PROGRAM Control
VAR


	ToggleSpiral: TOGGLE;
	HopperLevel_High: TON;
	HopperLevelHigh: BOOL;
	HopperLevelLow: BOOL;
	HopperLevelISLow: BOOL;
	HopperLevelISHigh: BOOL;
	Hopper_Level: Hopper_Level;
	Hopper_LevelLow: TON;
	Twin_Auger_Level: Hopper_Level;
	FRA3_HopperLevel_INT: INT;
	sSpice_Tank_Valve: BOOL;
	PreBrine_Delay: TON;
	PreBrineValveTON: TON;
	PreBrineValveTOF: TOF;
	Feed: ton;
	Auger: ton;
	FeedAugerResume: ton;
	Resume: BOOL;
	Auger_Resume: BOOL;
	HopperResume: tof;
	FillerCPM: FillerCPM_Current;
	sFillerCPM_Current: REAL;
	HopperLevelLow_Timer: TIME;
	SpareTON_1: TON;
END_VAR
VAR PERSISTENT
	SpareTONTest: BOOL;
	SpareTimerTest: BOOL;
	HopperLevelLowHMI: INT;
	HopperLevelLowCalc: INT;
	HopperLevelHighHMI: INT;
	HopperLevelHighCalc: INT;
	HopperLevelHigh_Timer: TIME;
	FeedAugerResumeHMI: INT;
	FeedAugerResumeCalc: INT;
	FeedAugerDelayHMITimer: TIME;
	sCloserJam_1_RealValue: REAL;
	sCloserJam_1RV: REAL;
	sCloserJam_1PT: TIME;
	sCloserJam_2_RealValue: REAL;
	sCloserJam_2RV: REAL;
	sCloserJam_2PT: TIME;
	sElevatorJam_RealValue: REAL;
	sElevatorJamRV: REAL;
	sElevatorJamPT: TIME;
	sFullCanBeltDelay_RealValue: REAL;
	sFullCanBeltDelayRV: REAL;
	sFullCanBeltDelayPT: TIME;
	sNoEmptyCansDelay_RealValue: REAL;
	sNoEmptyCansDelayRV: REAL;
	sNoEmptyCansDelayPT: TIME;
	sPrebrineFlapON_RealValue: REAL;
	sPrebrineFlapOFFRV: REAL;
	sPrebrineFlapONRV: REAL;
	sPrebrineFlapONPT: TIME;
	sPrebrineFlapOFF_RealValue: REAL;
	sPrebrineFlapOFFPT: TIME;
	sPrebrineValveON_RealValue: REAL;
	sPrebrineValveONRV: REAL;
	sPrebrineValveONPT: TIME;
	sPrebrineValveOFF_RealValue: REAL;
	sPrebrineValveOffRV: REAL;
	sPrebrineValveOffPT: TIME;
	sRefillJuicer_RealValue: REAL;
	sRefillJuicerRV: REAL;
	sRefillJuicerPT: TIME;
	sLowSpiceDisable_RealValue: REAL;
	sLowSpiceDisableRV: REAL;
	sLowSpiceDisablePT: TIME;
END_VAR
VAR // added by the converter: edge detectors and wires of the graphical bodies
    _w1, _w2, _w3 : BOOL;
END_VAR

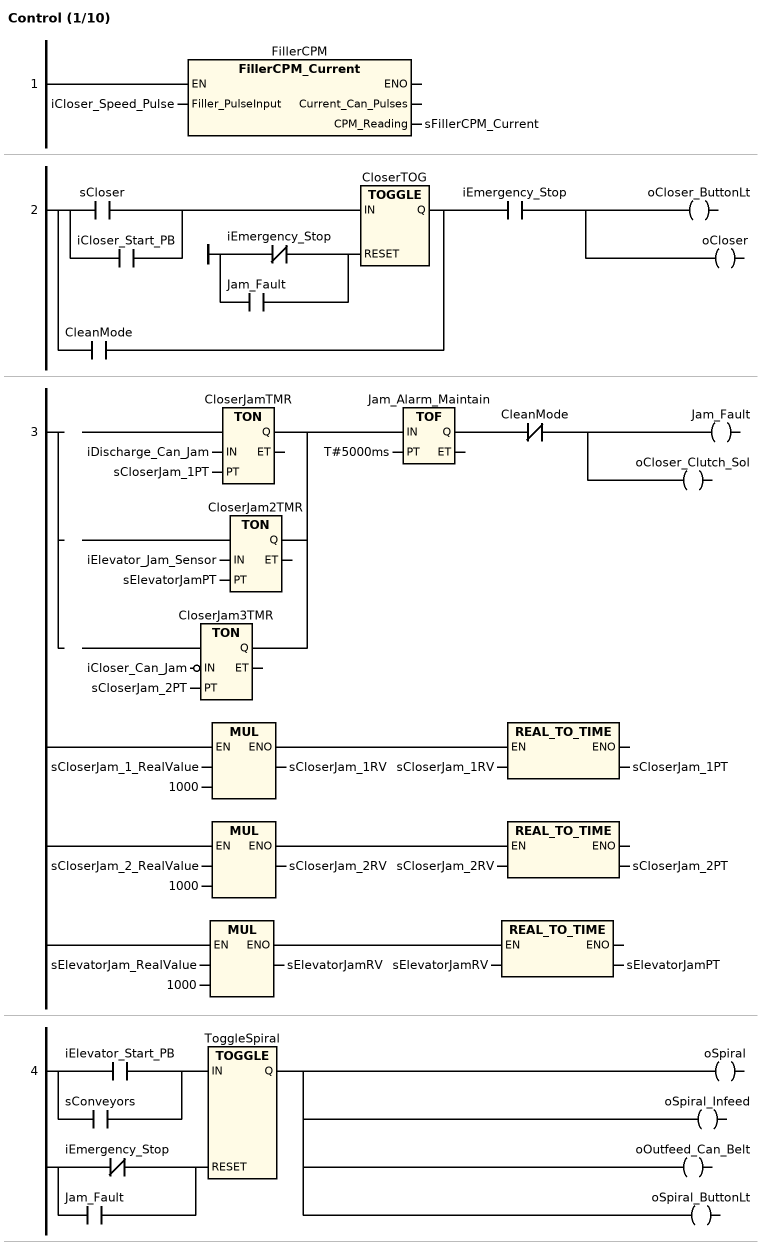
// NETWORK 1
FillerCPM(Filler_PulseInput := iCloser_Speed_Pulse, CPM_Reading => sFillerCPM_Current); // FillerCPM_Current

// NETWORK 2
CloserTOG(IN := sCloser OR iCloser_Start_PB, RESET := NOT iEmergency_Stop OR Jam_Fault); // TOGGLE
_w1 := (CloserTOG.Q OR CleanMode) AND iEmergency_Stop;
oCloser_ButtonLt := _w1;
oCloser := _w1;

// NETWORK 3
CloserJamTMR(IN := iDischarge_Can_Jam, PT := sCloserJam_1PT); // TON
CloserJam2TMR(IN := iElevator_Jam_Sensor, PT := sElevatorJamPT); // TON
CloserJam3TMR(IN := NOT iCloser_Can_Jam, PT := sCloserJam_2PT); // TON
Jam_Alarm_Maintain(IN := CloserJamTMR.Q OR CloserJam2TMR.Q OR CloserJam3TMR.Q, PT := T#5000ms); // TOF
_w2 := Jam_Alarm_Maintain.Q AND NOT CleanMode;
Jam_Fault := _w2;
oCloser_Clutch_Sol := _w2;
sCloserJam_1RV := sCloserJam_1_RealValue * 1000;
sCloserJam_1PT := REAL_TO_TIME(sCloserJam_1RV);
sCloserJam_2RV := sCloserJam_2_RealValue * 1000;
sCloserJam_2PT := REAL_TO_TIME(sCloserJam_2RV);
sElevatorJamRV := sElevatorJam_RealValue * 1000;
sElevatorJamPT := REAL_TO_TIME(sElevatorJamRV);

// NETWORK 4
ToggleSpiral(IN := iElevator_Start_PB OR sConveyors, RESET := NOT iEmergency_Stop OR Jam_Fault); // TOGGLE
oSpiral := ToggleSpiral.Q;
oSpiral_Infeed := ToggleSpiral.Q;
oOutfeed_Can_Belt := ToggleSpiral.Q;
oSpiral_ButtonLt := ToggleSpiral.Q;

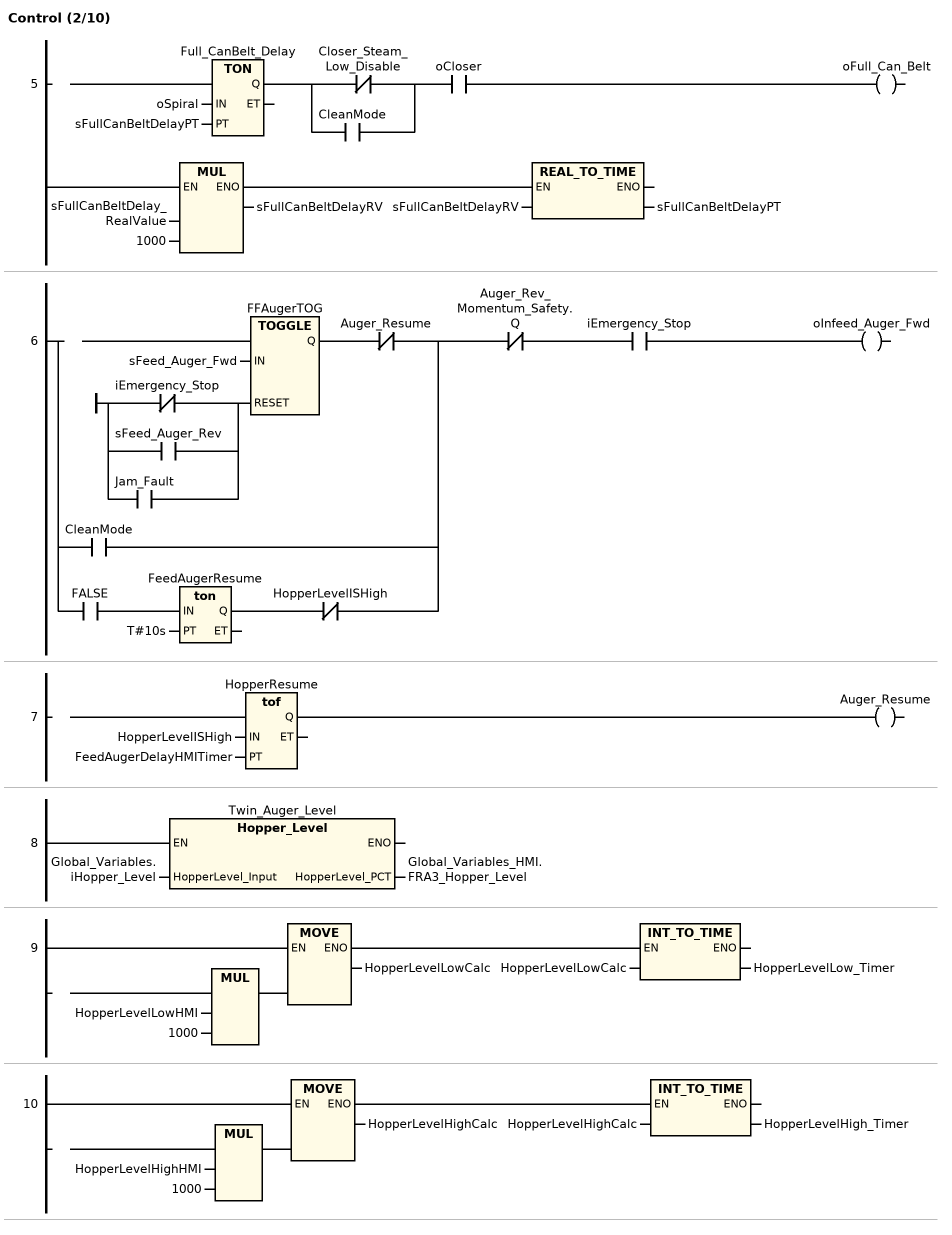
// NETWORK 5
Full_CanBelt_Delay(IN := oSpiral, PT := sFullCanBeltDelayPT); // TON
oFull_Can_Belt := Full_CanBelt_Delay.Q AND (NOT Closer_Steam_Low_Disable OR CleanMode) AND oCloser;
sFullCanBeltDelayRV := sFullCanBeltDelay_RealValue * 1000;
sFullCanBeltDelayPT := REAL_TO_TIME(sFullCanBeltDelayRV);

// NETWORK 6
FFAugerTOG(IN := sFeed_Auger_Fwd, RESET := NOT iEmergency_Stop OR sFeed_Auger_Rev OR Jam_Fault); // TOGGLE
FeedAugerResume(IN := FALSE, PT := T#10s); // ton
oInfeed_Auger_Fwd := (FFAugerTOG.Q AND NOT Auger_Resume OR CleanMode OR FeedAugerResume.Q AND NOT HopperLevelISHigh) AND NOT Auger_Rev_Momentum_Safety.Q AND iEmergency_Stop;

// NETWORK 7
HopperResume(IN := HopperLevelISHigh, PT := FeedAugerDelayHMITimer); // tof
Auger_Resume := HopperResume.Q;

// NETWORK 8
Twin_Auger_Level(HopperLevel_Input := Global_Variables.iHopper_Level, HopperLevel_PCT => Global_Variables_HMI.FRA3_Hopper_Level); // Hopper_Level

// NETWORK 9
HopperLevelLowCalc := HopperLevelLowHMI * 1000;
HopperLevelLow_Timer := INT_TO_TIME(HopperLevelLowCalc);

// NETWORK 10
HopperLevelHighCalc := HopperLevelHighHMI * 1000;
HopperLevelHigh_Timer := INT_TO_TIME(HopperLevelHighCalc);

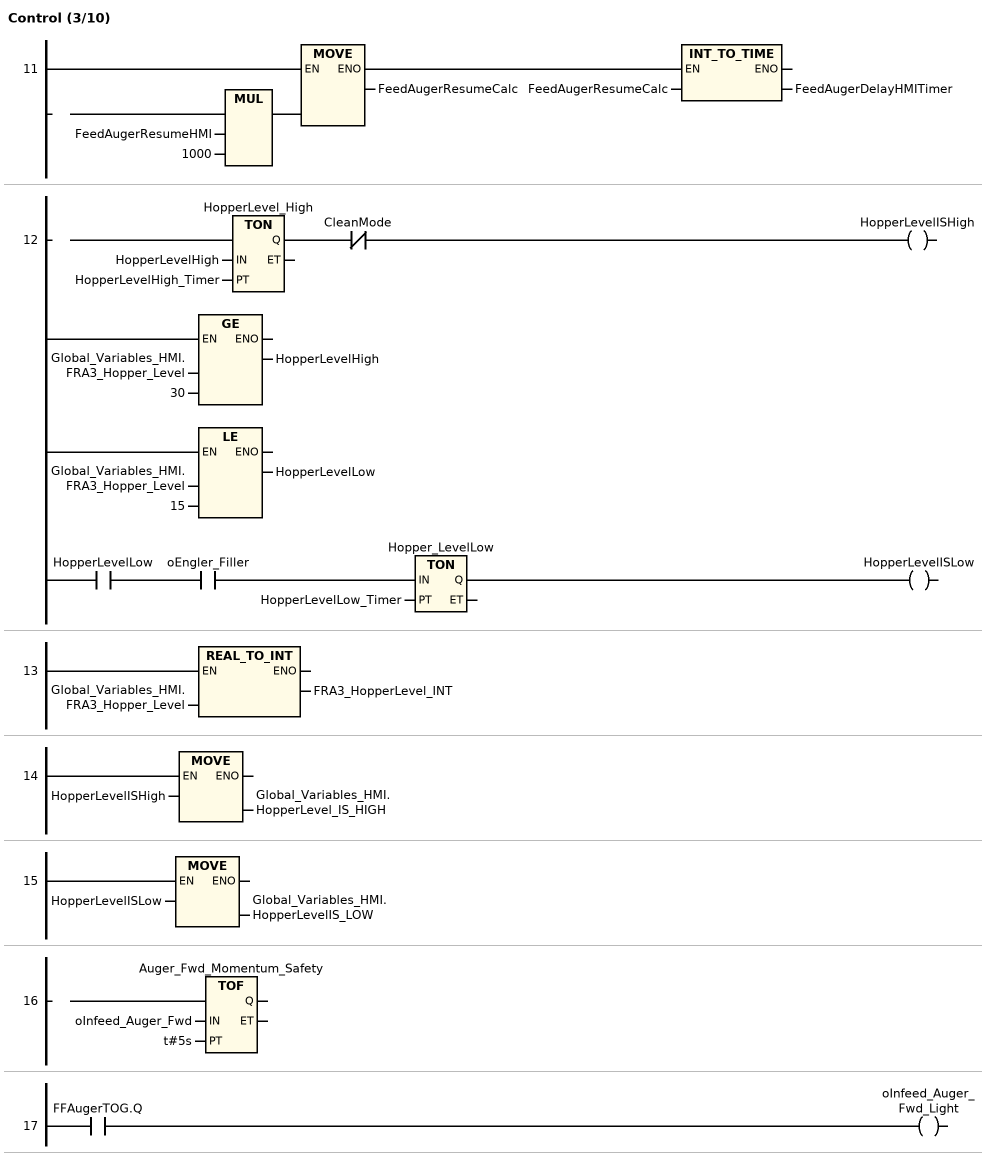
// NETWORK 11
FeedAugerResumeCalc := FeedAugerResumeHMI * 1000;
FeedAugerDelayHMITimer := INT_TO_TIME(FeedAugerResumeCalc);

// NETWORK 12
HopperLevel_High(IN := HopperLevelHigh, PT := HopperLevelHigh_Timer); // TON
HopperLevelISHigh := HopperLevel_High.Q AND NOT CleanMode;
HopperLevelHigh := Global_Variables_HMI.FRA3_Hopper_Level >= 30;
HopperLevelLow := Global_Variables_HMI.FRA3_Hopper_Level <= 15;
Hopper_LevelLow(IN := HopperLevelLow AND oEngler_Filler, PT := HopperLevelLow_Timer); // TON
HopperLevelISLow := Hopper_LevelLow.Q;

// NETWORK 13
FRA3_HopperLevel_INT := REAL_TO_INT(Global_Variables_HMI.FRA3_Hopper_Level);

// NETWORK 14
Global_Variables_HMI.HopperLevel_IS_HIGH := HopperLevelISHigh;

// NETWORK 15
Global_Variables_HMI.HopperLevelIS_LOW := HopperLevelISLow;

// NETWORK 16
Auger_Fwd_Momentum_Safety(IN := oInfeed_Auger_Fwd, PT := t#5s); // TOF

// NETWORK 17
oInfeed_Auger_Fwd_Light := FFAugerTOG.Q;

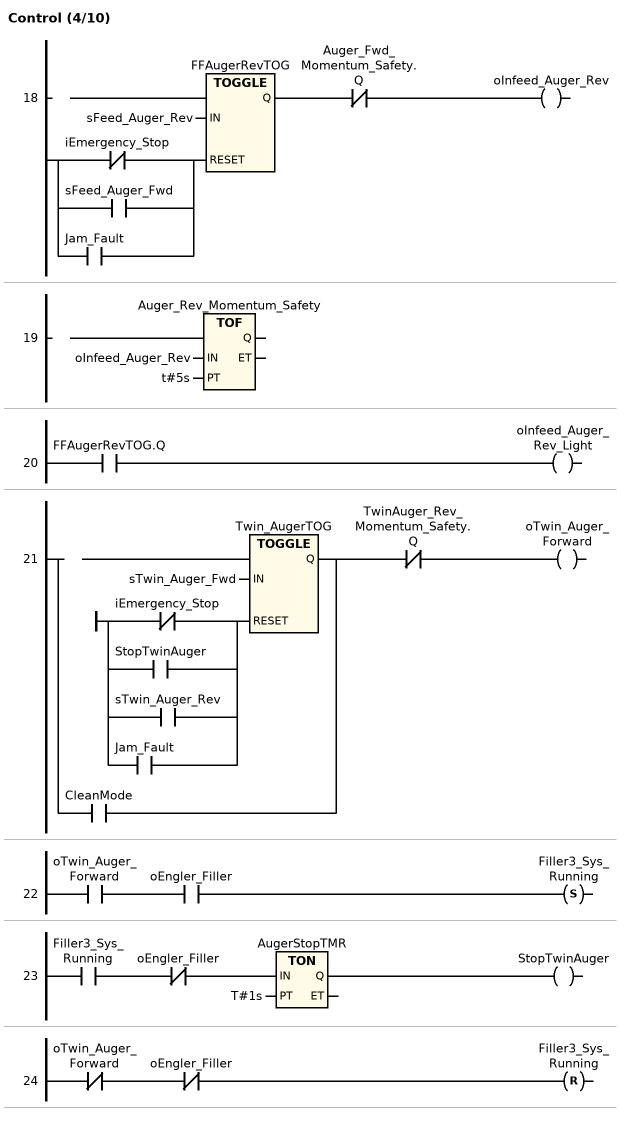
// NETWORK 18
FFAugerRevTOG(IN := sFeed_Auger_Rev, RESET := NOT iEmergency_Stop OR sFeed_Auger_Fwd OR Jam_Fault); // TOGGLE
oInfeed_Auger_Rev := FFAugerRevTOG.Q AND NOT Auger_Fwd_Momentum_Safety.Q;

// NETWORK 19
Auger_Rev_Momentum_Safety(IN := oInfeed_Auger_Rev, PT := t#5s); // TOF

// NETWORK 20
oInfeed_Auger_Rev_Light := FFAugerRevTOG.Q;

// NETWORK 21
Twin_AugerTOG(IN := sTwin_Auger_Fwd, RESET := NOT iEmergency_Stop OR StopTwinAuger OR sTwin_Auger_Rev OR Jam_Fault); // TOGGLE
oTwin_Auger_Forward := (Twin_AugerTOG.Q OR CleanMode) AND NOT TwinAuger_Rev_Momentum_Safety.Q;

// NETWORK 22
Filler3_Sys_Running S= oTwin_Auger_Forward AND oEngler_Filler;

// NETWORK 23
AugerStopTMR(IN := Filler3_Sys_Running AND NOT oEngler_Filler, PT := T#1s); // TON
StopTwinAuger := AugerStopTMR.Q;

// NETWORK 24
Filler3_Sys_Running R= NOT oTwin_Auger_Forward AND NOT oEngler_Filler;

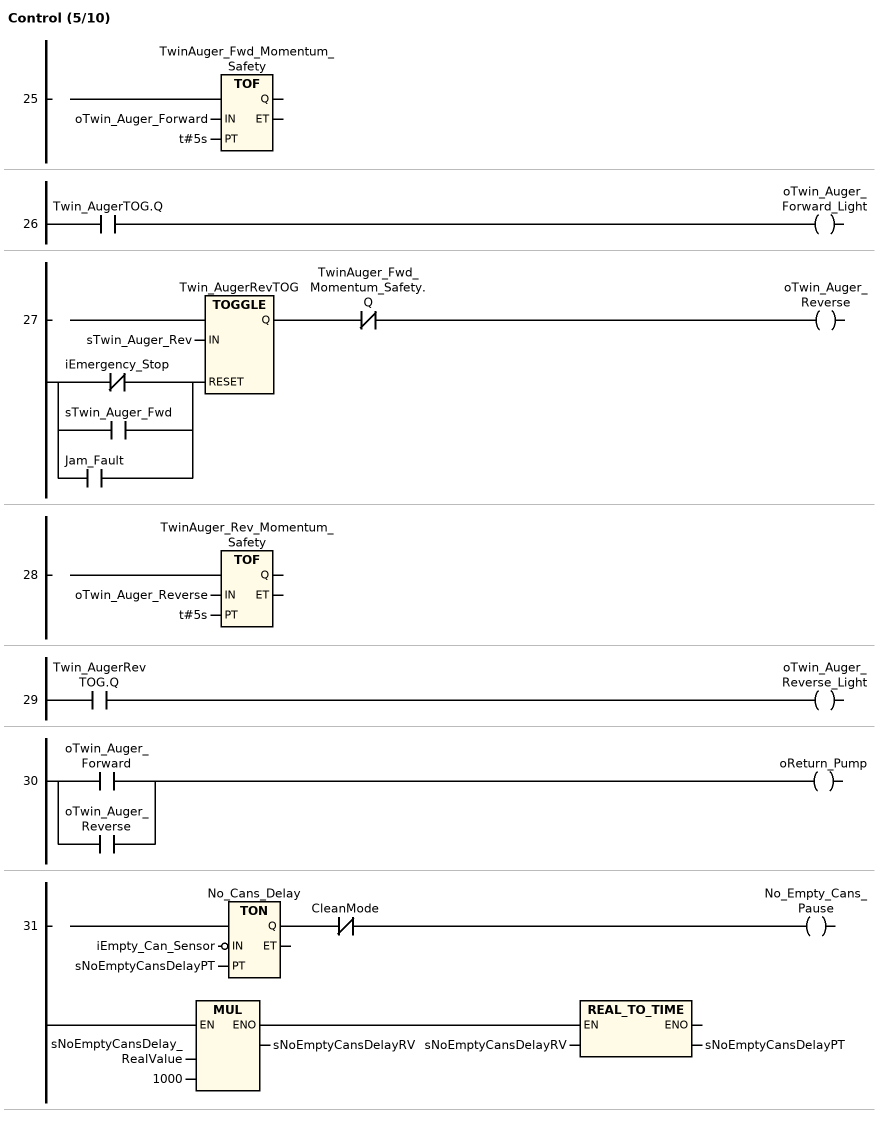
// NETWORK 25
TwinAuger_Fwd_Momentum_Safety(IN := oTwin_Auger_Forward, PT := t#5s); // TOF

// NETWORK 26
oTwin_Auger_Forward_Light := Twin_AugerTOG.Q;

// NETWORK 27
Twin_AugerRevTOG(IN := sTwin_Auger_Rev, RESET := NOT iEmergency_Stop OR sTwin_Auger_Fwd OR Jam_Fault); // TOGGLE
oTwin_Auger_Reverse := Twin_AugerRevTOG.Q AND NOT TwinAuger_Fwd_Momentum_Safety.Q;

// NETWORK 28
TwinAuger_Rev_Momentum_Safety(IN := oTwin_Auger_Reverse, PT := t#5s); // TOF

// NETWORK 29
oTwin_Auger_Reverse_Light := Twin_AugerRevTOG.Q;

// NETWORK 30
oReturn_Pump := oTwin_Auger_Forward OR oTwin_Auger_Reverse;

// NETWORK 31
No_Cans_Delay(IN := NOT iEmpty_Can_Sensor, PT := sNoEmptyCansDelayPT); // TON
No_Empty_Cans_Pause := No_Cans_Delay.Q AND NOT CleanMode;
sNoEmptyCansDelayRV := sNoEmptyCansDelay_RealValue * 1000;
sNoEmptyCansDelayPT := REAL_TO_TIME(sNoEmptyCansDelayRV);

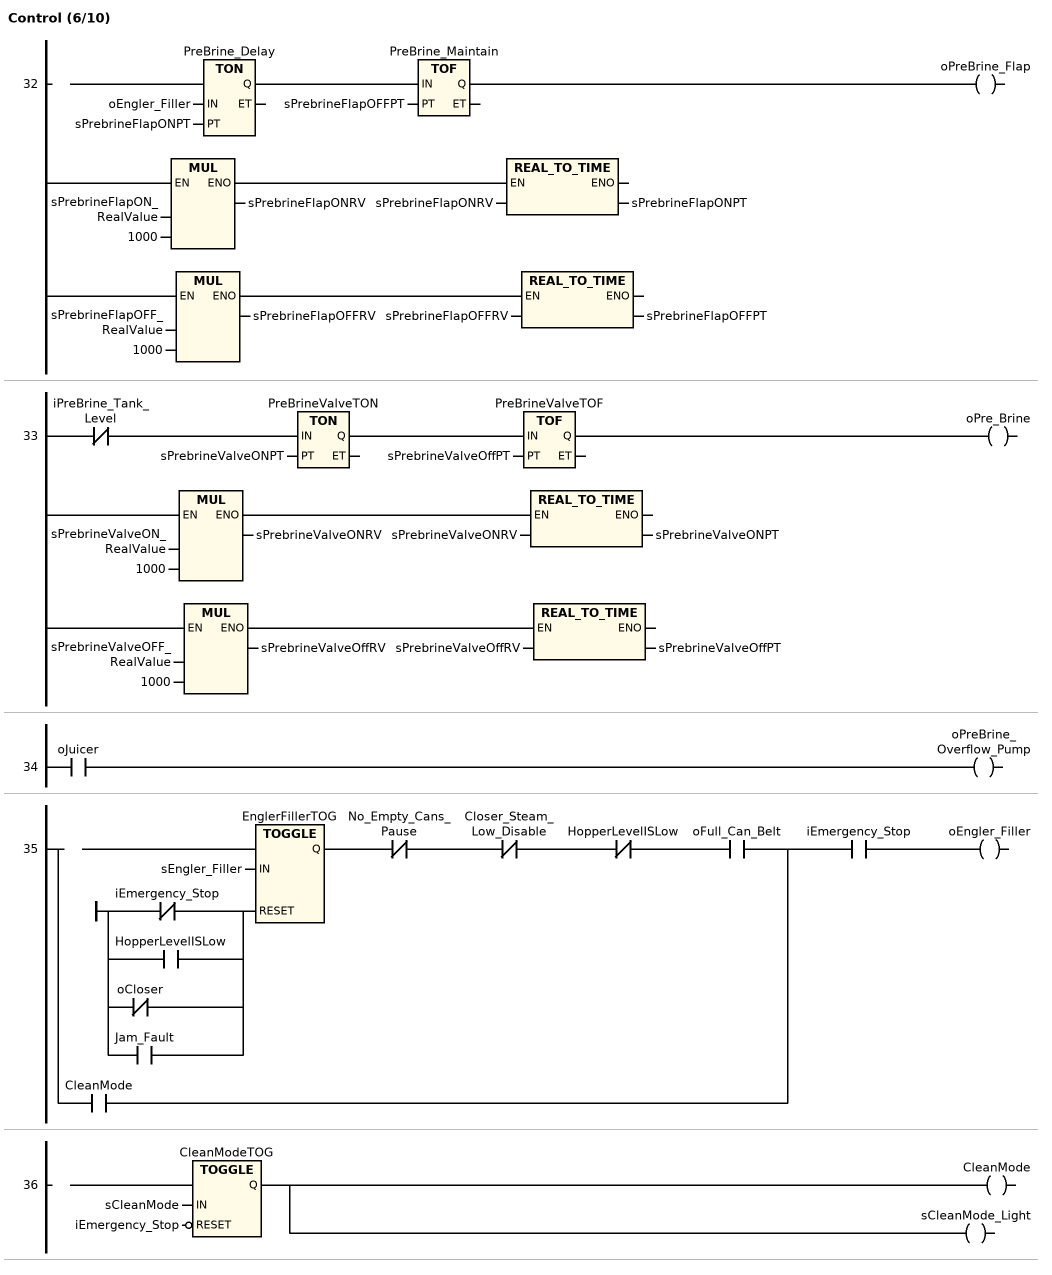
// NETWORK 32
PreBrine_Delay(IN := oEngler_Filler, PT := sPrebrineFlapONPT); // TON
PreBrine_Maintain(IN := PreBrine_Delay.Q, PT := sPrebrineFlapOFFPT); // TOF
oPreBrine_Flap := PreBrine_Maintain.Q;
sPrebrineFlapONRV := sPrebrineFlapON_RealValue * 1000;
sPrebrineFlapONPT := REAL_TO_TIME(sPrebrineFlapONRV);
sPrebrineFlapOFFRV := sPrebrineFlapOFF_RealValue * 1000;
sPrebrineFlapOFFPT := REAL_TO_TIME(sPrebrineFlapOFFRV);

// NETWORK 33
PreBrineValveTON(IN := NOT iPreBrine_Tank_Level, PT := sPrebrineValveONPT); // TON
PreBrineValveTOF(IN := PreBrineValveTON.Q, PT := sPrebrineValveOffPT); // TOF
oPre_Brine := PreBrineValveTOF.Q;
sPrebrineValveONRV := sPrebrineValveON_RealValue * 1000;
sPrebrineValveONPT := REAL_TO_TIME(sPrebrineValveONRV);
sPrebrineValveOffRV := sPrebrineValveOFF_RealValue * 1000;
sPrebrineValveOffPT := REAL_TO_TIME(sPrebrineValveOffRV);

// NETWORK 34
oPreBrine_Overflow_Pump := oJuicer;

// NETWORK 35
EnglerFillerTOG(IN := sEngler_Filler, RESET := NOT iEmergency_Stop OR HopperLevelISLow OR NOT oCloser OR Jam_Fault); // TOGGLE
oEngler_Filler := (EnglerFillerTOG.Q AND NOT No_Empty_Cans_Pause AND NOT Closer_Steam_Low_Disable AND NOT HopperLevelISLow AND oFull_Can_Belt OR CleanMode) AND iEmergency_Stop;

// NETWORK 36
CleanModeTOG(IN := sCleanMode, RESET := NOT iEmergency_Stop); // TOGGLE
CleanMode := CleanModeTOG.Q;
sCleanMode_Light := CleanModeTOG.Q;

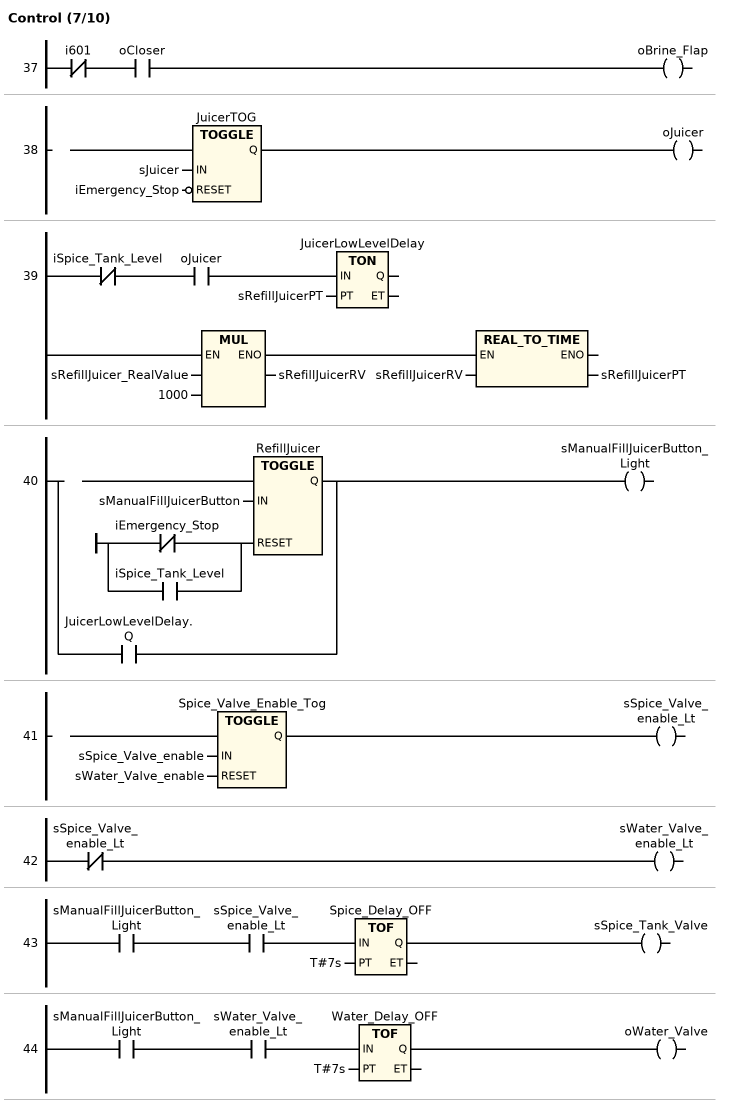
// NETWORK 37
oBrine_Flap := NOT i601 AND oCloser;

// NETWORK 38
JuicerTOG(IN := sJuicer, RESET := NOT iEmergency_Stop); // TOGGLE
oJuicer := JuicerTOG.Q;

// NETWORK 39
JuicerLowLevelDelay(IN := NOT iSpice_Tank_Level AND oJuicer, PT := sRefillJuicerPT); // TON
sRefillJuicerRV := sRefillJuicer_RealValue * 1000;
sRefillJuicerPT := REAL_TO_TIME(sRefillJuicerRV);

// NETWORK 40
RefillJuicer(IN := sManualFillJuicerButton, RESET := NOT iEmergency_Stop OR iSpice_Tank_Level); // TOGGLE
sManualFillJuicerButton_Light := RefillJuicer.Q OR JuicerLowLevelDelay.Q;

// NETWORK 41
Spice_Valve_Enable_Tog(IN := sSpice_Valve_enable, RESET := sWater_Valve_enable); // TOGGLE
sSpice_Valve_enable_Lt := Spice_Valve_Enable_Tog.Q;

// NETWORK 42
sWater_Valve_enable_Lt := NOT sSpice_Valve_enable_Lt;

// NETWORK 43
Spice_Delay_OFF(IN := sManualFillJuicerButton_Light AND sSpice_Valve_enable_Lt, PT := T#7s); // TOF
sSpice_Tank_Valve := Spice_Delay_OFF.Q;

// NETWORK 44
Water_Delay_OFF(IN := sManualFillJuicerButton_Light AND sWater_Valve_enable_Lt, PT := T#7s); // TOF
oWater_Valve := Water_Delay_OFF.Q;

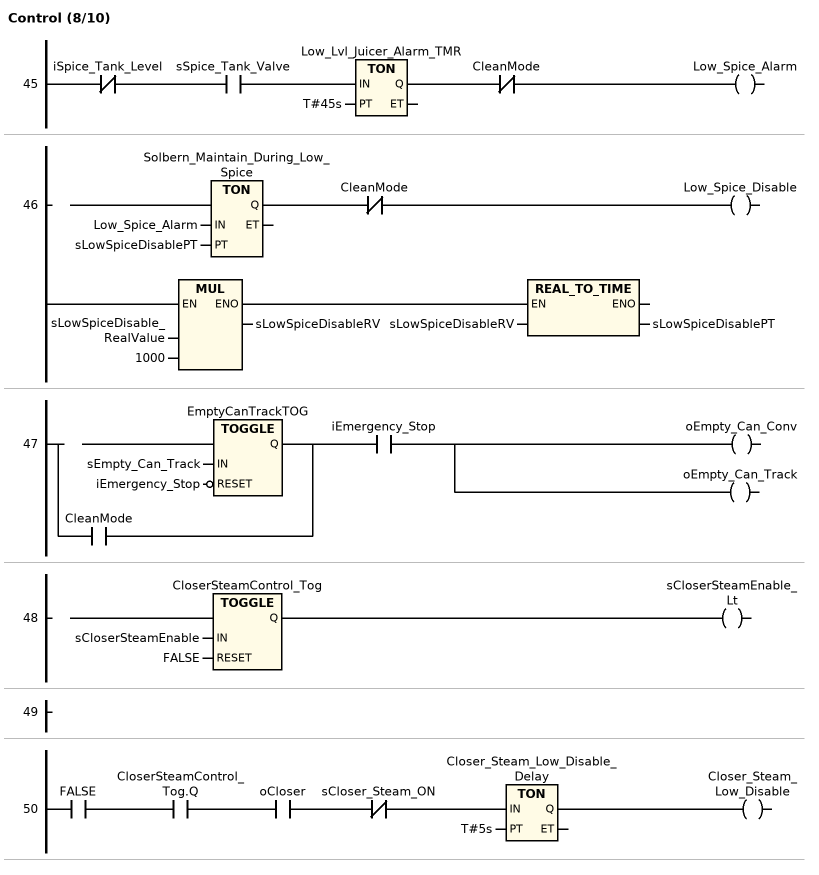
// NETWORK 45
Low_Lvl_Juicer_Alarm_TMR(IN := NOT iSpice_Tank_Level AND sSpice_Tank_Valve, PT := T#45s); // TON
Low_Spice_Alarm := Low_Lvl_Juicer_Alarm_TMR.Q AND NOT CleanMode;

// NETWORK 46
Solbern_Maintain_During_Low_Spice(IN := Low_Spice_Alarm, PT := sLowSpiceDisablePT); // TON
Low_Spice_Disable := Solbern_Maintain_During_Low_Spice.Q AND NOT CleanMode;
sLowSpiceDisableRV := sLowSpiceDisable_RealValue * 1000;
sLowSpiceDisablePT := REAL_TO_TIME(sLowSpiceDisableRV);

// NETWORK 47
EmptyCanTrackTOG(IN := sEmpty_Can_Track, RESET := NOT iEmergency_Stop); // TOGGLE
_w3 := (EmptyCanTrackTOG.Q OR CleanMode) AND iEmergency_Stop;
oEmpty_Can_Conv := _w3;
oEmpty_Can_Track := _w3;

// NETWORK 48
CloserSteamControl_Tog(IN := sCloserSteamEnable, RESET := FALSE); // TOGGLE
sCloserSteamEnable_Lt := CloserSteamControl_Tog.Q;

// NETWORK 49

// NETWORK 50
Closer_Steam_Low_Disable_Delay(IN := FALSE AND CloserSteamControl_Tog.Q AND oCloser AND NOT sCloser_Steam_ON, PT := T#5s); // TON
Closer_Steam_Low_Disable := Closer_Steam_Low_Disable_Delay.Q;

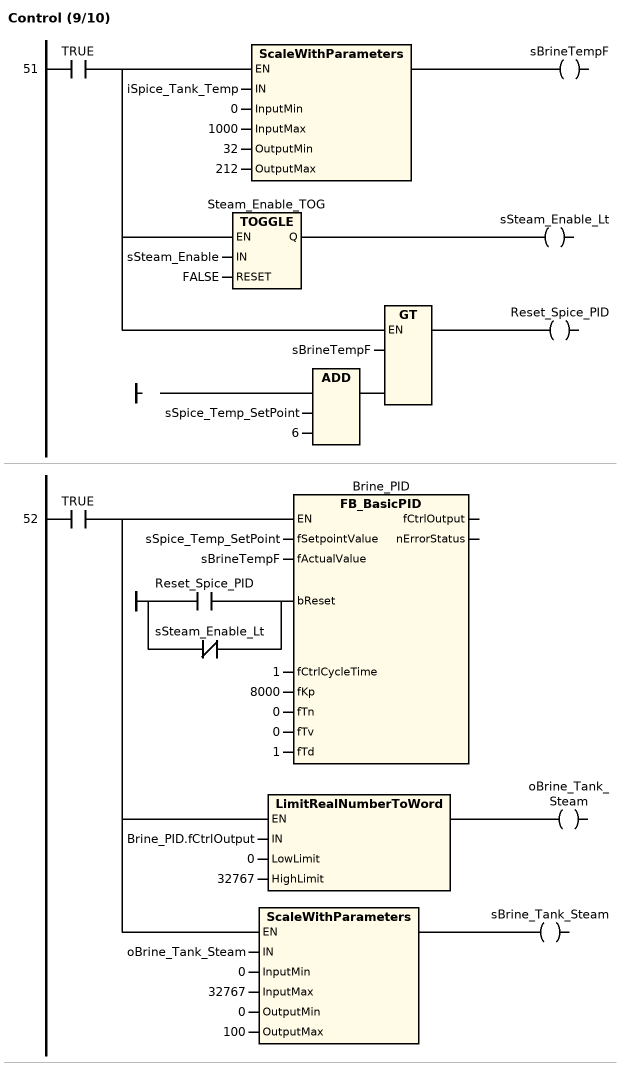
// NETWORK 51
sBrineTempF := ScaleWithParameters(IN := iSpice_Tank_Temp, InputMin := 0, InputMax := 1000, OutputMin := 32, OutputMax := 212);
Steam_Enable_TOG(IN := sSteam_Enable, RESET := FALSE); // TOGGLE
sSteam_Enable_Lt := Steam_Enable_TOG.Q;
Reset_Spice_PID := sBrineTempF > sSpice_Temp_SetPoint + 6;

// NETWORK 52
Brine_PID(
    fSetpointValue := sSpice_Temp_SetPoint,
    fActualValue := sBrineTempF,
    bReset := Reset_Spice_PID OR NOT sSteam_Enable_Lt,
    fCtrlCycleTime := 1,
    fKp := 8000,
    fTn := 0,
    fTv := 0,
    fTd := 1); // FB_BasicPID
oBrine_Tank_Steam := LimitRealNumberToWord(IN := Brine_PID.fCtrlOutput, LowLimit := 0, HighLimit := 32767);
sBrine_Tank_Steam := ScaleWithParameters(IN := oBrine_Tank_Steam, InputMin := 0, InputMax := 32767, OutputMin := 0, OutputMax := 100);

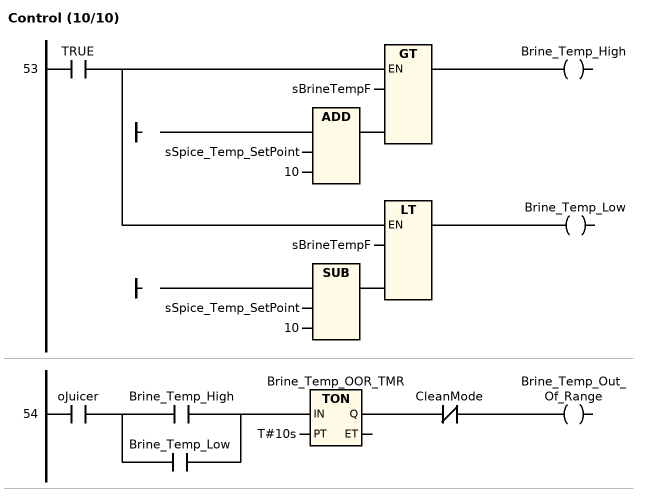
// NETWORK 53
Brine_Temp_High := sBrineTempF > sSpice_Temp_SetPoint + 10;
Brine_Temp_Low := sBrineTempF < sSpice_Temp_SetPoint - 10;

// NETWORK 54
Brine_Temp_OOR_TMR(IN := oJuicer AND (Brine_Temp_High OR Brine_Temp_Low), PT := T#10s); // TON
Brine_Temp_Out_Of_Range := Brine_Temp_OOR_TMR.Q AND NOT CleanMode;

END_PROGRAM

(* stored: Version 1.1.0.1, ProductVersion 3.1.4024.15
   POU Control: Id {b74eb2cb-e221-499c-b732-c095ade196eb}, SpecialFunc None *)
